// TIA Portal V18 export
TYPE "UDT_RTDadv"
// stored: IsFailsafeCompliant false
   STRUCT
      rValue : Real;   // Real value
      rFilterSet : Real;   // Filter value
      rCalibration : Real;   // Scale Min
      rDiv : Real := 100.0;   // Scale Max
      cFuncSystemID : Byte := 0;
      cFuncVar : Byte := 0;
      iReserv : Int;
   END_STRUCT;
END_TYPE
